INTERFACE I_AsynchronousRpcResponseFactory

METHOD PUBLIC TryCreate : BOOL
VAR_INPUT
	Destination : REFERENCE TO I_AsynchronousRpcResponse;
END_VAR
END_METHOD

END_INTERFACE

(* stored: Version 1.1.0.1, ProductVersion 3.1.4024.12
   Itf I_AsynchronousRpcResponseFactory: Id {ab248955-460c-0f24-2716-43d11523fb38}
   Method TryCreate: Id {464f5bb9-b0f7-0531-192b-1aca7824cae7} *)
